Fanuc KAREL source: ka00079.KL

PROGRAM KA00079
%NOLOCKGROUP
VAR
SRC : XYZWPREXT;DST : XYZWPREXT
BEGIN
--
SRC.X=1.0
DST=SRC
END KA00079
